PROGRAM MAIN
VAR
END_VAR

END_PROGRAM

(* stored: Version 1.1.0.1
   POU MAIN: Id {091d1eee-ce39-405b-b73c-640d90cd69e5} *)
